// TIA Portal V17 export
// export: Created 2023-12-01T06:57:26.8962748Z, ExportSetting None, DisplayName Totally Integrated Automation Portal, DisplayVersion V17 Update 5, DisplayName TIA Portal Openness, DisplayVersion V17 Update 5, DisplayName TIA Portal Teamcenter Gateway, DisplayVersion V17 Update 5, DisplayName TIA Portal Version Control Interface, DisplayVersion V17, DisplayName SINAMICS Startdrive Advanced, DisplayVersion V17, DisplayName SINAMICS Startdrive G130, G150, S120, S150, SINAMICS MV, S210, DisplayVersion V17, DisplayName SINAMICS Startdrive G110M, G120, G120C, G120D, G120P, G115D, DisplayVersion V17, DisplayName STEP 7 Professional, DisplayVersion V17 Update 5, DisplayName STEP 7 Safety, DisplayVersion V17, DisplayName WinCC Advanced / Unified PC, DisplayVersion V17 Update 5
DATA_BLOCK "Motor_aux"   // DB999
// stored: AutoNumber false, InstanceOfName SpinMotor_V0.1, InstanceOfType FB
"SpinMotor_V0.1"
   // VAR_INPUT
   //    BwdEn : Bool;
   //    "With Drive" : Bool;
   // END_VAR
   // VAR
   //    Auto : Bool;
   //    Man : Bool;
   //    ManStop : Bool;
   //    PowerOn : Bool;
   //    Overload : Bool;
   //    RepairSwitch : Bool;
   //    Overtemperature : Bool;
   //    Alm { S7_SetPoint := 'True'} : "UdtMotorsAlm_IM";
   //    FWD { S7_SetPoint := 'True'} : "UdtMotorsState_IM";
   //    BWD { S7_SetPoint := 'True'} : "UdtMotorsState_IM";
   //    Drive { S7_SetPoint := 'True'} : "UdtMotorDrive_IM";
   //    HMIStatus : "UdtMotorsHMIStatus_IM";
   //    HMICommand { S7_SetPoint := 'True'} : "UdtMotorsHMICommand_IM";
   // END_VAR
BEGIN
END_DATA_BLOCK
